// TIA Portal project "CTA_travail_Hugo_Uriel" (V19)

(* hardware
DEVICE "S7-300/ET200M station_1"  S7-300 station
   slot 0: "Rail_0"  Rail  6ES7 390-1***0-0AA0
   slot 2: "PLC_1"  CPU 314C-2 PN/DP  6ES7 314-6EH04-0AB0  V3.3
      slot 2: "PROFINET interface_1"  PN-IO
         slot 1: "Port_1"  Port
         slot 2: "Port_2"  Port
      slot 5: "DI 24/DO 16_1"  DI24/DO16
      slot 6: "AI 5/AO 2_1"  AI5/AO2
      slot 7: "Count_1"  Counter
      slot 8: "Positioning_1"  Positioning
*)

// ===== PLC "PLC_1"  CPU 314C-2 PN/DP =====

VAR_GLOBAL   // PLC tag table "Variables Station Separating"
   "PART_AV" AT %I0.0 : Bool;   // Pièce Disponible
   "B2" AT %I0.1 : Bool;   // Présence pièce pour analyxe
   "B3" AT %I0.2 : Bool;   // Vérification profondeur pièce
   "B4" AT %I0.3 : Bool;   // Vérin rotatif rentré
   "B5" AT %I0.4 : Bool;   // Convoyeur 2 plein
   "B6" AT %I0.5 : Bool;   // Pièce en sortie de station
   "IP_FI_B" AT %I0.6 : Bool;   // Simulation station suivante libre
   "IP_FI" AT %I0.7 : Bool;   // Station suivante libre
   "BP Start" AT %I1.0 : Bool;   // NO Départ cycle
   "BP Stop" AT %I1.1 : Bool;   // NF Fin cycle
   "Selecteur Auto/Manu" AT %I1.2 : Bool;   // Choix mode fonctionnement
   "BP Reset" AT %I1.3 : Bool;   // Initialisation station
   "Emergency Stop" AT %I1.5 : Bool;   // Arrêt d'urgence (ponté)
   "M1" AT %Q0.0 : Bool;   // Convoyeur principal - Marche
   "M2" AT %Q0.1 : Bool;   // Convoyeur secondaire - Marche
   "1M1" AT %Q0.2 : Bool;   // Blocage pièce - sorti au repos
   "2M1" AT %Q0.3 : Bool;   // Aiguillage - convoyeur secondaire
   "IP_N_FO" AT %Q0.7 : Bool;   // Station occupée
   "LStart" AT %Q1.0 : Bool;   // Lampe BP Start
   "LReset" AT %Q1.1 : Bool;   // Lampe BP Reset
   "Q1" AT %Q1.2 : Bool;   // Voyant lumineux Gauche
   "Q2" AT %Q1.3 : Bool;   // Voyant lumineux Droite
   "B3 Analogique" AT %IW800 : Int;   // Profondeur piece
END_VAR

VAR_GLOBAL   // PLC tag table "Default tag table"
   "RETVAL WW" AT %MW80 : Int;
END_VAR

DATA_BLOCK "Data_block_memo"   // DB1
{ S7_Optimized_Access := 'FALSE' }
VERSION : 0.1
   VAR
      memo_convoyeur_1 : Bool;
      memo_convoyeur_2 : Bool;
      memo_verrin_aiguillage : Bool;
      memo_verrin_blocage : Bool;
      IN_Avancer_Tapis_1 : Bool;
      IN_Avancer_Tapis_2 : Bool;
      IN_Verrin_blocage : Bool;
      IN_Verrin_aiguillage : Bool;
      OUT_position_verrin_aiguillage : Bool;
      OUT_position_verrin_blocage : Bool;
      valeur_profondeur : Real;
      rent_val_capteur : Word;
      auto : Bool;
      manu : Bool;
      marche : Bool;
      arret : Bool;
      profondeur : Bool;
   END_VAR
BEGIN
END_DATA_BLOCK

DATA_BLOCK "Tapis_roulant_DB_1"   // DB2
{ S7_Optimized_Access := 'FALSE' }
VERSION : 0.1
// stored: InstanceOfName Tapis_roulant_DB
"Tapis_roulant_DB"
BEGIN
END_DATA_BLOCK

DATA_BLOCK "Tapis_roulant_DB_2"   // DB3
{ S7_Optimized_Access := 'FALSE' }
VERSION : 0.1
// stored: InstanceOfName Tapis_roulant_DB
"Tapis_roulant_DB"
BEGIN
END_DATA_BLOCK

DATA_BLOCK "Verrin_DB_Aiguillage"   // DB4
{ S7_Optimized_Access := 'FALSE' }
VERSION : 0.1
// stored: InstanceOfName Verrin_DB
"Verrin_DB"
BEGIN
END_DATA_BLOCK

DATA_BLOCK "Verrin_DB_blocage"   // DB5
{ S7_Optimized_Access := 'FALSE' }
VERSION : 0.1
// stored: InstanceOfName Verrin_DB
"Verrin_DB"
BEGIN
END_DATA_BLOCK

// folder: SystemBlocksFolder/ReportSystemErrorFolder

DATA_BLOCK "RSE_DIAGNOSTIC_STATUS_DB"   // DB127
TITLE = Report System Error Diagnostic Block
{ S7_Optimized_Access := 'FALSE' }
AUTHOR : SIMATIC
FAMILY : RSEDIAG
NAME : RSE7
VERSION : 1.0
// This DB is part of report system error and will be updated by the RSE FB.
//  It is an interface for support of system diagnosis via the CPU web server.
   VAR
      Directory : Struct
         D_Version : Word := WORD#16#0100;   // Version that supports RSE
         D_pGlobalState : Word := WORD#16#0010;   // Byte offset to the start of the "GlobalState" section
         D_pQuery : Word := WORD#16#0014;   // Byte offset to the start of the "Query" section
         D_pComponent : Word := WORD#16#0020;   // Byte offset to the start of the "Component" section
         D_pError : Word := WORD#16#0024;   // Byte offset to the start of the "Error" section
         D_pState : Word := WORD#16#0028;   // Byte offset to the start of the "State" section
         D_pAlarm : Word := WORD#16#005A;   // Byte offset to the start of the "Alarm" section
         D_pSubComponent : Word := WORD#16#0082;   // Byte offset to the start of the "Subcomponent" section
      END_STRUCT;
      GlobalState : Struct
         G_EventCount : Word;   // ID of the last event (counter)
         G_StartReporting : Bool;   // Startup evaluation running
      END_STRUCT;
      Query : Struct
         Q_ClientID_User : DWord;   // ID of the client
         Q_ClientID_Intern : DWord;   // ID of the client (internal)
         Q_WithSubComponent : Bool;   // With/without status of the underlying components (slower)
         Q_SubComponentAlarm : Bool;   // AS-iMaster gibt AS-iSlave Alarme zurück
         Q_Reserved2 : Bool;   // Reserved
         Q_Reserved3 : Bool;   // Reserved
         Q_Reserved4 : Bool;   // Reserved
         Q_Reserved5 : Bool;   // Reserved
         Q_Reserved6 : Bool;   // Reserved
         Q_Reserved7 : Bool;   // Reserved
         Q_Start : Bool;   // Start query
         Q_Error : Byte;   // Internal error in query
         Q_Reserved8 : Byte;   // Reserved
      END_STRUCT;
      Component : Struct
         C_AddressMode : Byte;   // Addressing mode of the module
         C_Reserved1 : Byte;   // Reserved
         C_ComponentID : Word;   // Hardware ID of the component (internal)
      END_STRUCT;
      Error : Struct
         E_ErrorNo : Word;   // Index of the requested/actual error
         E_LastError : Bool;   // TRUE, if E_ErrorNo contains the indes of the last error, otherwise FALSE
      END_STRUCT;
      State : Struct
         S_Hierarchy : Byte;   // Reserved
         S_Periphery : Byte;   // Reserved
         S_SupFault : Bool;   // The component is not obtainable
         S_NotAvailable : Bool;   // The component does not exist
         S_Faulty : Bool;   // The component is disrupted; the "Alarm" section is not empty
         S_MoreErrors : Bool;   // There are more errors than RSE can store.
         S_Maintenance1 : Bool;   // Maintenance required is indicated
         S_Maintenance2 : Bool;   // Maintenance demand is indicated
         S_Deactivated : Bool;   // The component was deactivated
         S_Reserved2 : Bool;   // Reserved
         S_SubFault : Bool;   // An underlying component is disrupted
         S_SubMaintenance1 : Bool;   // Maintenance required is indicated for an underlying component
         S_SubMaintenance2 : Bool;   // Maintenance demand is indicated for an underlying component
         S_SubDeactivated : Bool;   // At least one lower-level component is disabled
         S_Reserved4 : Bool;   // Reserved
         S_Reserved5 : Bool;   // Reserved
         S_Reserved6 : Bool;   // Reserved
         S_Reserved7 : Bool;   // Reserved
         S_TIAMS : DWord;   // Maintenance state of the component
         S_TIAMSChannelExist : DWord;   // Maintenance state: Configured channels
         S_TIAMSChannelOK : DWord;   // Maintenance State: Disrupted channels
         S_ChannelCount : Word;   // Number of channels; Valid only when Q_WithSubComponent is set
         S_ChannelVector : Array[0..255] of Bool;   // List of channels involved; Valid only when Q_WithSubComponent is set
      END_STRUCT;
      Alarm : Struct
         A_ComponentID : Word;   // Hardware ID of the component (internal)
         A_TextID1 : Word;   // ID of the first error text
         A_TextLexikonID1 : Word;   // ID of the first error text lexicon
         A_HelpTextLexikonID1 : Word;   // ID of the first help text lexicon
         A_MapTextID : Word;   // ID of the first error text in the export file (HMI)
         A_MapHelpTextID : Word;   // ID of the first help text in the export file (HMI)
         A_TextID2 : Word;   // ID of the second error text
         A_TextLexikonID2 : Word;   // ID of the second error text lexicon
         A_HelpTextLexikonID2 : Word;   // ID of the second help text lexicon
         A_MapTextID2 : Word;   // ID of the second error text in the export file (HMI)
         A_MapHelpTextID2 : Word;   // ID of the second help text in the export file (HMI)
         A_AlarmID : DWord;   // Message number
         A_ValueCount : Word := WORD#16#000C;   // Number of other occupied bytes
         A_AssociatedValue : Array[1..6] of Word;   // Associated values of the message
      END_STRUCT;
      SubComponent : Struct
         U_SubComponentCount : Word;   // Number of underlying components
         U_SubComponentFault : Array[1..8] of Byte;   // List of status of subordinate components, 1 byte per component
      END_STRUCT;
   END_VAR
BEGIN
END_DATA_BLOCK

// folder: (top level)

FUNCTION_BLOCK "Verrin_DB"   // FB1, FBD
{ S7_Optimized_Access := 'FALSE' }
VERSION : 0.1
   VAR_INPUT
      Activation : Bool;
      Positon : Bool;
   END_VAR
   VAR_OUTPUT
      Marche : Bool;
      Position_retour : Bool;
   END_VAR
BEGIN

REGION Network 1
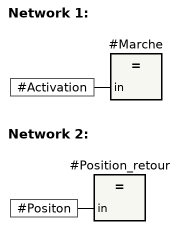
   #Marche := #Activation;
END_REGION

REGION Network 2
   #Position_retour := #Positon;
END_REGION
END_FUNCTION_BLOCK

FUNCTION_BLOCK "Tapis_roulant_DB"   // FB2, FBD
{ S7_Optimized_Access := 'FALSE' }
VERSION : 0.1
   VAR_INPUT
      Start_Avant : Bool;
   END_VAR
   VAR_OUTPUT
      Run : Bool;
   END_VAR
   VAR_TEMP
      moteur_tapis : Bool;
   END_VAR
BEGIN

REGION Network 1
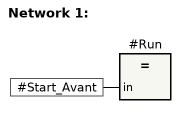
   #Run := #Start_Avant;
END_REGION
END_FUNCTION_BLOCK

FUNCTION "Mode_auto" : Void   // FC1, FBD
{ S7_Optimized_Access := 'FALSE' }
VERSION : 0.1
   VAR_TEMP
      State : Int;
      Mode_auto : Bool;
   END_VAR
   VAR_TEMP   // added for the SCL form of the ladder/FBD networks
      _w1 : Bool;
   END_VAR
BEGIN

REGION Network 1
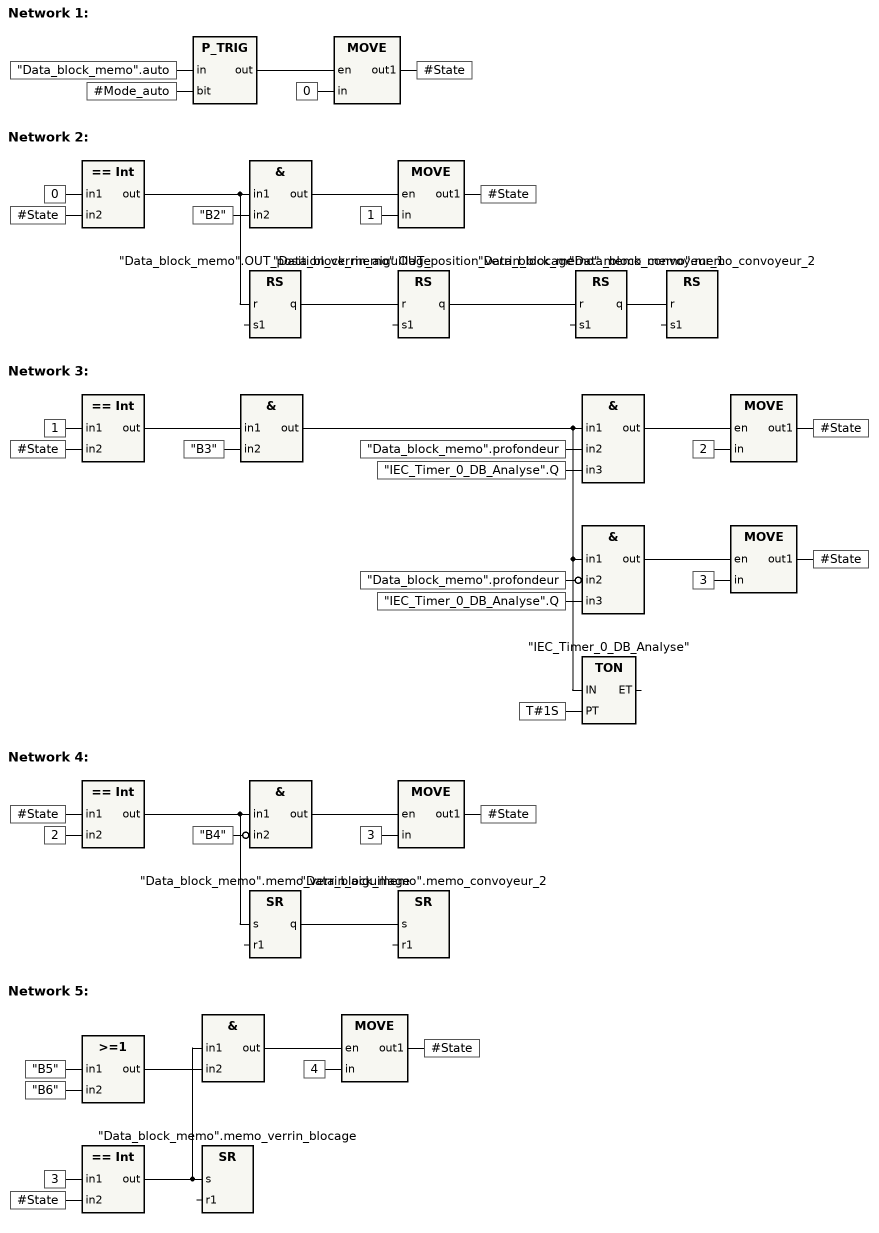
   #_w1 := "Data_block_memo".auto AND NOT #Mode_auto;   // rising edge
   #Mode_auto := "Data_block_memo".auto;
   IF #_w1 THEN #State := 0; END_IF;
END_REGION

REGION Network 2
   #_w1 := 0 = #State;
   IF #_w1 AND "B2" THEN #State := 1; END_IF;
   IF #_w1 THEN
       "Data_block_memo".OUT_position_verrin_aiguillage := FALSE;   // RS flip-flop
   END_IF;
   IF "Data_block_memo".OUT_position_verrin_aiguillage THEN
       "Data_block_memo".OUT_position_verrin_blocage := FALSE;   // RS flip-flop
   END_IF;
   IF "Data_block_memo".OUT_position_verrin_blocage THEN
       "Data_block_memo".memo_convoyeur_1 := FALSE;   // RS flip-flop
   END_IF;
   IF "Data_block_memo".memo_convoyeur_1 THEN
       "Data_block_memo".memo_convoyeur_2 := FALSE;   // RS flip-flop
   END_IF;
END_REGION

REGION Network 3
   #_w1 := (1 = #State) AND "B3";
   IF #_w1 AND "Data_block_memo".profondeur AND "IEC_Timer_0_DB_Analyse".Q THEN #State := 2; END_IF;
   IF #_w1 AND NOT "Data_block_memo".profondeur AND "IEC_Timer_0_DB_Analyse".Q THEN #State := 3; END_IF;
   "IEC_Timer_0_DB_Analyse".TON(IN := #_w1, PT := T#1S);
END_REGION

REGION Network 4
   #_w1 := #State = 2;
   IF #_w1 AND NOT "B4" THEN #State := 3; END_IF;
   IF #_w1 THEN
       "Data_block_memo".memo_verrin_aiguillage := TRUE;   // SR flip-flop
   END_IF;
   IF "Data_block_memo".memo_verrin_aiguillage THEN
       "Data_block_memo".memo_convoyeur_2 := TRUE;   // SR flip-flop
   END_IF;
END_REGION

REGION Network 5
   #_w1 := 3 = #State;
   IF #_w1 AND ("B5" OR "B6") THEN #State := 4; END_IF;
   IF #_w1 THEN
       "Data_block_memo".memo_verrin_blocage := TRUE;   // SR flip-flop
   END_IF;
END_REGION

REGION Network 6
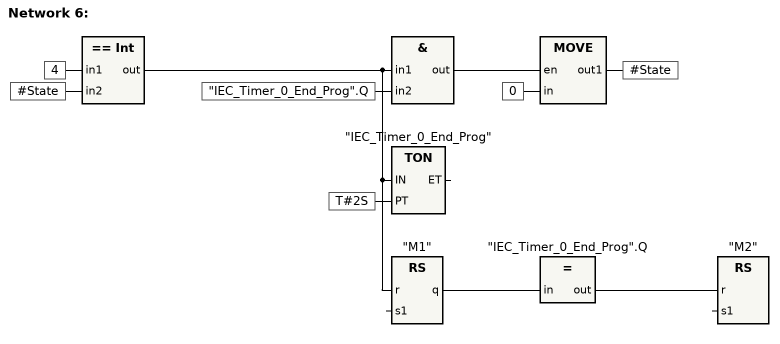
   #_w1 := 4 = #State;
   IF #_w1 AND "IEC_Timer_0_End_Prog".Q THEN #State := 0; END_IF;
   "IEC_Timer_0_End_Prog".TON(IN := #_w1, PT := T#2S);
   IF #_w1 THEN
       "M1" := FALSE;   // RS flip-flop
   END_IF;
   "IEC_Timer_0_End_Prog".Q := "M1";
   IF "M1" THEN
       "M2" := FALSE;   // RS flip-flop
   END_IF;
END_REGION
END_FUNCTION

FUNCTION "WebServeur" : Void   // FC2, LAD
{ S7_Optimized_Access := 'FALSE' }
VERSION : 0.1
BEGIN

REGION Network 1
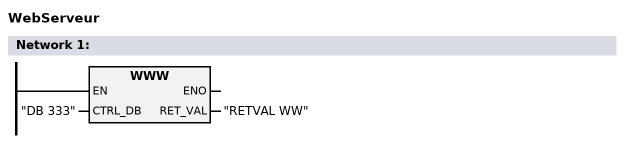
   "RETVAL WW" := WWW(CTRL_DB := "DB 333");
END_REGION
END_FUNCTION

FUNCTION "Lecteure/Ecriture_analogique" : Void   // FC3, FBD
{ S7_Optimized_Access := 'FALSE' }
VERSION : 0.1
   VAR_INPUT
      Valeur_IN : Int;
   END_VAR
   VAR_OUTPUT
      Valeur_OUT : Real;
      Ret_val_1 : Word;
   END_VAR
   VAR_TEMP
      Mem_Valeur_out : Real;
   END_VAR
   VAR CONSTANT
      Bipolar : Bool;
   END_VAR
BEGIN

REGION Network 1
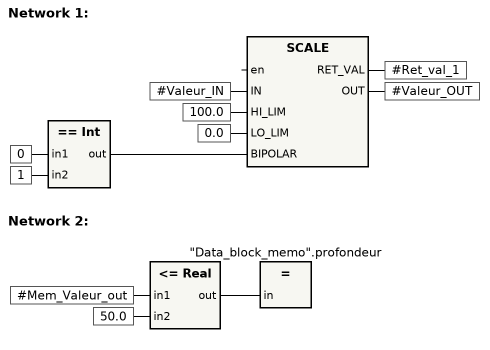
   #Ret_val_1 := SCALE(IN := #Valeur_IN, HI_LIM := 100.0, LO_LIM := 0.0, BIPOLAR := 0 = 1, OUT => #Valeur_OUT);
END_REGION

REGION Network 2
   "Data_block_memo".profondeur := #Mem_Valeur_out <= 50.0;
END_REGION
END_FUNCTION

FUNCTION "Mode-focntionnement" : Void   // FC4, FBD
{ S7_Optimized_Access := 'FALSE' }
VERSION : 0.1
   VAR_INPUT
      "Auto/Manu" : Bool;
      Start : Bool;
      Stop : Bool;
      Reset : Bool;
   END_VAR
   VAR_OUTPUT
      Auto_out : Bool;
      Manu_out : Bool;
      Mode_marche : Bool;
      Mode_arret : Bool;
   END_VAR
   VAR_TEMP
      marche_mem : Bool;
      P_trig_changement : Bool;
      P_trig_changement_1 : Bool;
      false : Bool;
      Arret_mem : Bool;
   END_VAR
BEGIN

REGION Network 1
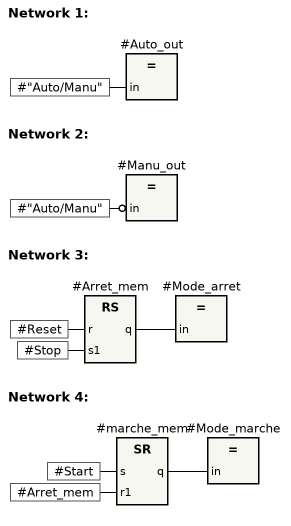
   #Auto_out := #"Auto/Manu";
END_REGION

REGION Network 2
   #Manu_out := NOT #"Auto/Manu";
END_REGION

REGION Network 3
   IF #Reset THEN
       #Arret_mem := FALSE;   // RS flip-flop
   END_IF;
   IF #Stop THEN #Arret_mem := TRUE; END_IF;
   #Mode_arret := #Arret_mem;
END_REGION

REGION Network 4
   IF #Start THEN
       #marche_mem := TRUE;   // SR flip-flop
   END_IF;
   IF #Arret_mem THEN #marche_mem := FALSE; END_IF;
   #Mode_marche := #marche_mem;
END_REGION
END_FUNCTION

FUNCTION "mode_manu" : Void   // FC5, FBD
{ S7_Optimized_Access := 'FALSE' }
VERSION : 0.1
BEGIN

REGION Network 1: Tapis 1
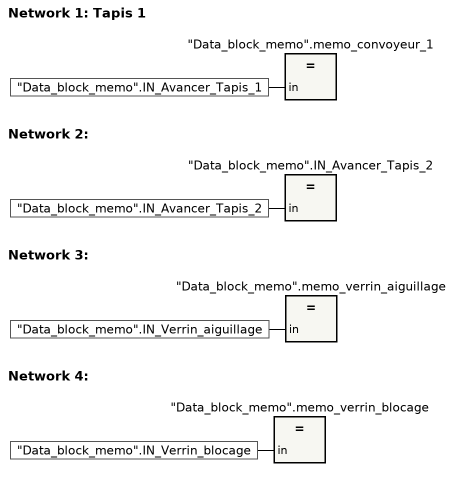
   "Data_block_memo".memo_convoyeur_1 := "Data_block_memo".IN_Avancer_Tapis_1;
END_REGION

REGION Network 2
   "Data_block_memo".IN_Avancer_Tapis_2 := "Data_block_memo".IN_Avancer_Tapis_2;
END_REGION

REGION Network 3
   "Data_block_memo".memo_verrin_aiguillage := "Data_block_memo".IN_Verrin_aiguillage;
END_REGION

REGION Network 4
   "Data_block_memo".memo_verrin_blocage := "Data_block_memo".IN_Verrin_blocage;
END_REGION
END_FUNCTION

ORGANIZATION_BLOCK "Main"   // OB1, LAD
TITLE = "Main Program Sweep (Cycle)"
{ S7_Optimized_Access := 'FALSE' }
VERSION : 0.1
   VAR_TEMP
      OB1_EV_CLASS : Byte;   // Bits 0-3 = 1 (Coming event), Bits 4-7 = 1 (Event class 1)
      OB1_SCAN_1 : Byte;   // 1 (Cold restart scan 1 of OB 1), 3 (Scan 2-n of OB 1)
      OB1_PRIORITY : Byte;   // Priority of OB Execution
      OB1_OB_NUMBR : Byte;   // 1 (Organization block 1, OB1)
      OB1_RESERVED_1 : Byte;   // Reserved for system
      OB1_RESERVED_2 : Byte;   // Reserved for system
      OB1_PREV_CYCLE : Int;   // Cycle time of previous OB1 scan (milliseconds)
      OB1_MIN_CYCLE : Int;   // Minimum cycle time of OB1 (milliseconds)
      OB1_MAX_CYCLE : Int;   // Maximum cycle time of OB1 (milliseconds)
      OB1_DATE_TIME : Date_And_Time;   // Date and time OB1 started
   END_VAR
BEGIN

REGION Network 1
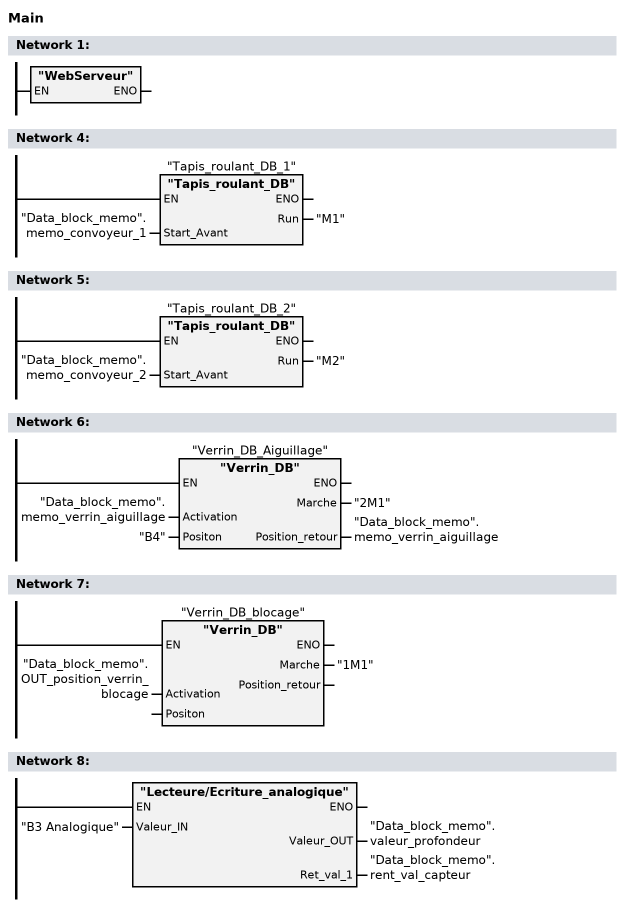
   RUNG wire#powerrail
      "WebServeur"()
   END_RUNG
   // the same network as SCL:
   "WebServeur"();
END_REGION

REGION Network 4
   RUNG wire#powerrail
      "Tapis_roulant_DB_1"(Start_Avant := "Data_block_memo".memo_convoyeur_1, Run => "M1")
   END_RUNG
   // the same network as SCL:
   "Tapis_roulant_DB_1"(Start_Avant := "Data_block_memo".memo_convoyeur_1, Run => "M1");   // "Tapis_roulant_DB"
END_REGION

REGION Network 5
   RUNG wire#powerrail
      "Tapis_roulant_DB_2"(Start_Avant := "Data_block_memo".memo_convoyeur_2, Run => "M2")
   END_RUNG
   // the same network as SCL:
   "Tapis_roulant_DB_2"(Start_Avant := "Data_block_memo".memo_convoyeur_2, Run => "M2");   // "Tapis_roulant_DB"
END_REGION

REGION Network 6
   RUNG wire#powerrail
      "Verrin_DB_Aiguillage"(Activation := "Data_block_memo".memo_verrin_aiguillage, Positon := "B4", Marche => "2M1", Position_retour => "Data_block_memo".memo_verrin_aiguillage)
   END_RUNG
   // the same network as SCL:
   "Verrin_DB_Aiguillage"(Activation := "Data_block_memo".memo_verrin_aiguillage,   // "Verrin_DB"
                          Positon := "B4",
                          Marche => "2M1",
                          Position_retour => "Data_block_memo".memo_verrin_aiguillage);
END_REGION

REGION Network 7
   RUNG wire#powerrail
      "Verrin_DB_blocage"(Activation := "Data_block_memo".OUT_position_verrin_blocage, Positon :=, Marche => "1M1", Position_retour =>)
   END_RUNG
   // the same network as SCL:
   "Verrin_DB_blocage"(Activation := "Data_block_memo".OUT_position_verrin_blocage, Marche => "1M1");   // "Verrin_DB"
END_REGION

REGION Network 8
   RUNG wire#powerrail
      "Lecteure/Ecriture_analogique"(Valeur_IN := "B3 Analogique", Valeur_OUT => "Data_block_memo".valeur_profondeur, Ret_val_1 => "Data_block_memo".rent_val_capteur)
   END_RUNG
   // the same network as SCL:
   "Lecteure/Ecriture_analogique"(Valeur_IN := "B3 Analogique",
                           Valeur_OUT => "Data_block_memo".valeur_profondeur,
                           Ret_val_1 => "Data_block_memo".rent_val_capteur);
END_REGION

REGION Network 10 (STL): Call system diagnostics block
         CALL  "RSE_FB", "RSE_DB";
END_REGION
END_ORGANIZATION_BLOCK

ORGANIZATION_BLOCK "I/O_FLT1"   // OB82, STL
TITLE = "I/O Point Fault"
{ S7_Optimized_Access := 'FALSE' }
VERSION : 0.1
   VAR_TEMP
      OB82_EV_CLASS : Byte;   // 16#39, Event class 3, Entering event state, Internal fault event
      OB82_FLT_ID : Byte;   // 16#XX, Fault identifcation code
      OB82_PRIORITY : Byte;   // Priority of OB Execution
      OB82_OB_NUMBR : Byte;   // 82 (Organization block 82, OB82)
      OB82_RESERVED_1 : Byte;   // Reserved for system
      OB82_IO_FLAG : Byte;   // Input (01010100), Output (01010101)
      OB82_MDL_ADDR : Word;   // Base address of module with fault
      OB82_MDL_DEFECT : Bool;   // Module defective
      OB82_INT_FAULT : Bool;   // Internal fault
      OB82_EXT_FAULT : Bool;   // External fault
      OB82_PNT_INFO : Bool;   // Point information
      OB82_EXT_VOLTAGE : Bool;   // External voltage low
      OB82_FLD_CONNCTR : Bool;   // Field wiring connector missing
      OB82_NO_CONFIG : Bool;   // Module has no configuration data
      OB82_CONFIG_ERR : Bool;   // Module has configuration error
      OB82_MDL_TYPE : Byte;   // Type of module
      OB82_SUB_MDL_ERR : Bool;   // Sub-Module is missing or has error
      OB82_COMM_FAULT : Bool;   // Communication fault
      OB82_MDL_STOP : Bool;   // Module is stopped
      OB82_WTCH_DOG_FLT : Bool;   // Watch dog timer stopped module
      OB82_INT_PS_FLT : Bool;   // Internal power supply fault
      OB82_PRIM_BATT_FLT : Bool;   // Primary battery is in fault
      OB82_BCKUP_BATT_FLT : Bool;   // Backup battery is in fault
      OB82_RESERVED_2 : Bool;   // Reserved for system
      OB82_RACK_FLT : Bool;   // Rack fault, only for bus interface module
      OB82_PROC_FLT : Bool;   // Processor fault
      OB82_EPROM_FLT : Bool;   // EPROM fault
      OB82_RAM_FLT : Bool;   // RAM fault
      OB82_ADU_FLT : Bool;   // ADU fault
      OB82_FUSE_FLT : Bool;   // Fuse fault
      OB82_HW_INTR_FLT : Bool;   // Hardware interupt input in fault
      OB82_RESERVED_3 : Bool;   // Reserved for system
      OB82_DATE_TIME : Date_And_Time;   // Date and time OB82 started
   END_VAR
BEGIN

REGION Network 1: Call system diagnostics block
         CALL  "RSE_FB", "RSE_DB";
END_REGION
END_ORGANIZATION_BLOCK

ORGANIZATION_BLOCK "I/O_FLT2"   // OB83, STL
TITLE = "I/O Point Fault"
{ S7_Optimized_Access := 'FALSE' }
VERSION : 0.1
   VAR_TEMP
      OB83_EV_CLASS : Byte;   // 16#38/39, Event class 3, module inserted/removed (8/9)
      OB83_FLT_ID : Byte;   // 16#XX, Fault identifcation code
      OB83_PRIORITY : Byte;   // Priority of OB Execution
      OB83_OB_NUMBR : Byte;   // 83 (Organization block 83, OB83)
      OB83_RESERVED_1 : Byte;   // Reserved for system
      OB83_MDL_ID : Byte;   // Input module (01010100), Output module (01010101)
      OB83_MDL_ADDR : Word;   // Base address of module with point fault
      OB83_RACK_NUM : Int;   // Number of rack that has module with point fault
      OB83_MDL_TYPE : Word;   // Module type with point fault
      OB83_DATE_TIME : Date_And_Time;   // Date and time OB83 started
   END_VAR
BEGIN

REGION Network 1: Call system diagnostics block
         CALL  "RSE_FB", "RSE_DB";
END_REGION
END_ORGANIZATION_BLOCK

ORGANIZATION_BLOCK "OBNL_FLT"   // OB85, STL
TITLE = "Organization Block (OB) Not Loaded Fault"
{ S7_Optimized_Access := 'FALSE' }
   VAR_TEMP
      OB85_EV_CLASS : Byte;   // 16#35 Event class 3
      OB85_FLT_ID : Byte;   // 16#XX, Fault identification code
      OB85_PRIORITY : Byte;   // Priority of OB Execution
      OB85_OB_NUMBR : Byte;   // 85 (Organization block 85, OB85)
      OB85_RESERVED_1 : Byte;   // Reserved for system
      OB85_RESERVED_2 : Byte;   // Reserved for system
      OB85_RESERVED_3 : Int;   // Reserved for system
      OB85_ERR_EV_CLASS : Byte;   // Class of event causing error
      OB85_ERR_EV_NUM : Byte;   // Number of event causing error
      OB85_OB_PRIOR : Byte;   // Priority of OB causing error
      OB85_OB_NUM : Byte;   // Number of OB causing error
      OB85_DATE_TIME : Date_And_Time;   // Date and time OB85 started
   END_VAR
BEGIN

REGION Network 1
         L     b#16#A1;  //
         L     #OB85_FLT_ID;
         ==I;
         JC    K_OB;
         L     b#16#A2;  //
         ==I;
         JC    K_OB;
         L     b#16#A3;  //
         L     #OB85_FLT_ID;
         ==I;
         JC    K_B;
         JU    F_PA;
END_REGION

REGION Network 2
   K_OB: JU    STOP;
         JU    ENDE;
END_REGION

REGION Network 3
   K_B:  JU    STOP;
         JU    ENDE;
END_REGION

REGION Network 4
   F_PA: NOP   0;
         JU    ENDE;
END_REGION

REGION Network 5
   STOP: CALL  STP;
END_REGION

REGION Network 6

   //

   ENDE: NOP   0;
END_REGION
END_ORGANIZATION_BLOCK

ORGANIZATION_BLOCK "RACK_FLT"   // OB86, STL
TITLE = "Loss Of Rack Fault"
{ S7_Optimized_Access := 'FALSE' }
VERSION : 0.1
   VAR_TEMP
      OB86_EV_CLASS : Byte;   // 16#38/39 Event class 3
      OB86_FLT_ID : Byte;   // 16#C1/C4/C5, Fault identification code
      OB86_PRIORITY : Byte;   // Priority of OB Execution
      OB86_OB_NUMBR : Byte;   // 86 (Organization block 86, OB86)
      OB86_RESERVED_1 : Byte;   // Reserved for system
      OB86_RESERVED_2 : Byte;   // Reserved for system
      OB86_MDL_ADDR : Word;   // Base address of IM module in rack with fault
      OB86_RACKS_FLTD : Array[0..31] of Bool;   // Racks in fault
      OB86_DATE_TIME : Date_And_Time;   // Date and time OB86 started
   END_VAR
BEGIN

REGION Network 1: Call system diagnostics block
         CALL  "RSE_FB", "RSE_DB";
END_REGION
END_ORGANIZATION_BLOCK